{attribute 'GeneratedUsingTerminal: EP4374-0002-0016'}
{attribute addProperty BoxType "EP4374-0002-0016"}
{attribute addProperty Description "EP4374-0002 2Ch. Ana. Input +/-10V, 0-10V, 0/4-20mA configurable; 2Ch. Ana. Output +/-10V, 0-10V, 0/4-20mA configurable"}
{attribute addProperty Physics "YY"}
{attribute addProperty Id "AI_TxPDO_Map_Standard_Channel_1AT %I*AI_TxPDO_Map_Standard_Channel_A8DF64E310AI_TxPDO_Map_Standard_Channel_2AT %I*AI_TxPDO_Map_Standard_Channel_A8DF64E310AO_RxPDO_Map_Channel_3AT %Q*AO_Output_Channel_BA7EBB7C2AO_RxPDO_Map_Channel_4AT %Q*AO_Output_Channel_BA7EBB7C2WcStateAT %I*WcState_9091E0EB2InfoDataAT %I*InfoData_32EB74EA10"}
{attribute addProperty CRC "3572113972"}
{attribute addProperty Size "36"}
TYPE EP4374_D4EA2234 EXTENDS EtcSlaveBoxBase_77A0E4A7 :
STRUCT
	{attribute addProperty Name "AI_TxPDO_Map_Standard_Channel_1"}
	AI_TxPDO_Map_Standard_Channel_1 : AI_TxPDO_Map_Standard_Channel_A8DF64E3;
	{attribute addProperty Name "AI_TxPDO_Map_Standard_Channel_2"}
	AI_TxPDO_Map_Standard_Channel_2 : AI_TxPDO_Map_Standard_Channel_A8DF64E3;
	{attribute addProperty Name "AO_RxPDO_Map_Channel_3"}
	AO_RxPDO_Map_Channel_3 : AO_Output_Channel_BA7EBB7C;
	{attribute addProperty Name "AO_RxPDO_Map_Channel_4"}
	AO_RxPDO_Map_Channel_4 : AO_Output_Channel_BA7EBB7C;
	{attribute addProperty Name "WcState"}
	WcState : WcState_9091E0EB;
	{attribute addProperty Name "InfoData"}
	InfoData : InfoData_32EB74EA;
END_STRUCT
END_TYPE

(* stored: Version 1.2.0.0, ProductVersion 3.1.4024.9
   DUT EP4374_D4EA2234: Id {14f07171-c4b3-46b6-bdb0-ce69f569b29e} *)
